# EPICS substitutions: db/ecmcEL3174_0to10V.substitutions
file ecmcEcSlave.template
{
    pattern {}
            {}
}

#Actually the scalinging is between 0..10.737V (see manual)
file ecmcEL3XXX-chX.template
{
	pattern {CH_ID, LINR,    ESLO,             EOFF,   EGU,        PREC, LOW, LOLO,  HIGH,  HIHI,    HYST, LLSV,    LSV,     HSV,     HHSV   }
    		{1,     "SLOPE", 3.2767723624E-4,  0,      "V",        3,    0,   -1,    10,    10.5,    0,    "MAJOR", "MINOR", "MINOR", "MAJOR"}
	    	{2,     "SLOPE", 3.2767723624E-4,  0,      "V",        3,    0,   -1,    10,    10.5,    0,    "MAJOR", "MINOR", "MINOR", "MAJOR"}
		    {3,     "SLOPE", 3.2767723624E-4,  0,      "V",        3,    0,   -1,    10,    10.5,    0,    "MAJOR", "MINOR", "MINOR", "MAJOR"}
		    {4,     "SLOPE", 3.2767723624E-4,  0,      "V",        3,    0,   -1,    10,    10.5,    0,    "MAJOR", "MINOR", "MINOR", "MAJOR"}

}
